Fanuc KAREL source: compact_preamble.KL

PROGRAM KF00115
%NOLOCKGROUP
VAR
I:INTEGER;J:INTEGER;X:REAL;Y:REAL;B:BOOLEAN;C:BOOLEAN;TXT : STRING[80];TXT2 : STRING[80];AI : ARRAY[4] OF INTEGER;BI : ARRAY[4] OF INTEGER;P : XYZWPR
JP : JOINTPOS9
PF : POSITION
V1 : VECTOR
V2 : VECTOR
STATUS:INTEGER
ROUTINE FADD(P1:INTEGER):INTEGER
BEGIN
RETURN((P1 + 1))
END FADD
BEGIN
I=FADD(2)
END KF00115
